PROGRAM P3_03_ProcessData
VAR
	stDBParam 					:ST_ProcessData;	
	fbDBWrite					:FB_PLCDBWriteEvt(sNetId:=CONST.AMS_NETID, tTimeout:=DEFAULT_ADS_TIMEOUT);
	tableColumns				:ARRAY [0..8] OF STRING(50) := ['batch', 'number', 'name', 'value1', 'value2', 'value3', 'value4', 'value5', 'value6'];
	arrParam					:ARRAY [0..8] OF ST_ExpParameter := [(sParaName := 'batch', nParaSize := 101, eParaType := E_EXPPARAMETERTYPE.STRING_),
															 (sParaName := 'number', nParaSize := 101, eParaType := E_EXPPARAMETERTYPE.STRING_),
															 (sParaName := 'name', nParaSize := 101, eParaType := E_EXPPARAMETERTYPE.STRING_),
															 (sParaName := 'value1', nParaSize := 101, eParaType := E_EXPPARAMETERTYPE.Float32), 
															 (sParaName := 'value2', nParaSize := 101, eParaType := E_EXPPARAMETERTYPE.Float32),
															 (sParaName := 'value3', nParaSize := 101, eParaType := E_EXPPARAMETERTYPE.Float32),
															 (sParaName := 'value4', nParaSize := 101, eParaType := E_EXPPARAMETERTYPE.Float32),
															 (sParaName := 'value5', nParaSize := 101, eParaType := E_EXPPARAMETERTYPE.Float32),
															 (sParaName := 'value6', nParaSize := 101, eParaType := E_EXPPARAMETERTYPE.Float32)];
	fbDeleteTable    			:FB_PLCDBCmdEvt(sNetID:=CONST.AMS_NETID, tTimeout:=DEFAULT_ADS_TIMEOUT);	
	sDelete						:STRING;	
	sDeleteAll					:STRING;
	sDeleteBatch				:STRING;
	bDelete						:BOOL;								 
	bWrite						:BOOL;		
	
	rChopper1Speed				:REAL;
	rChopper2Speed				:REAL;
END_VAR
VAR // added by the converter: edge detectors and wires of the graphical bodies
    _rt1, _rt2 : R_TRIG;
END_VAR

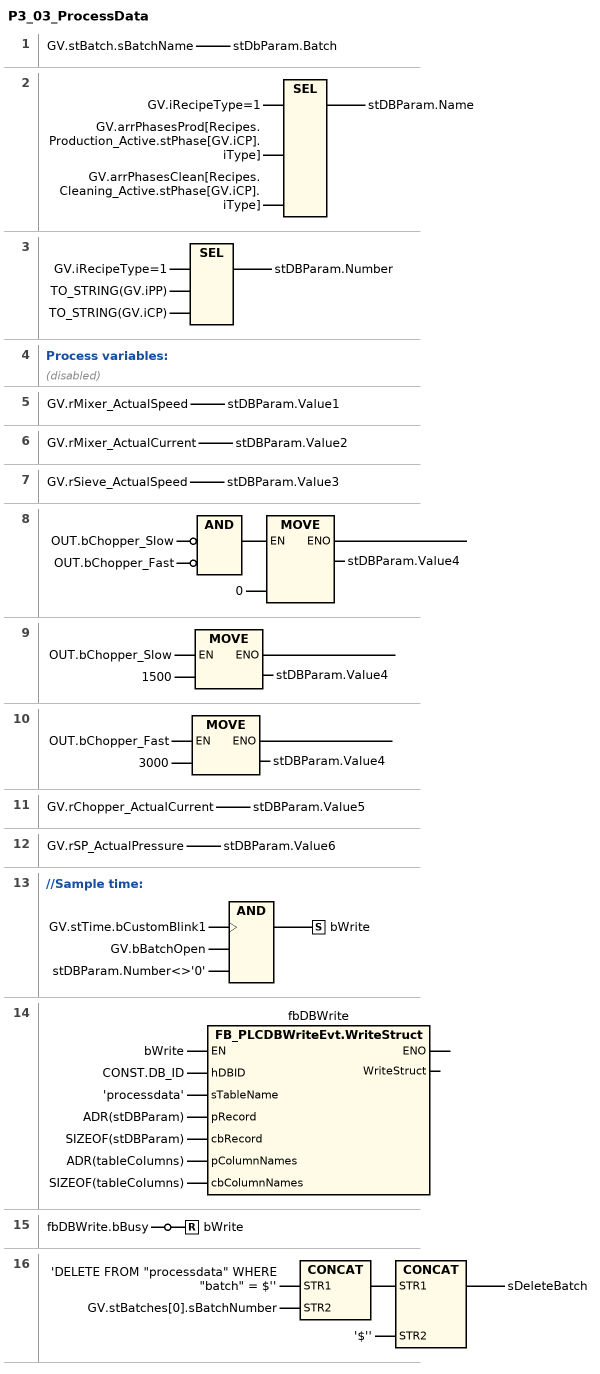
// NETWORK 1
stDbParam.Batch := GV.stBatch.sBatchName;

// NETWORK 2
stDBParam.Name := SEL(GV.iRecipeType=1, GV.arrPhasesProd[Recipes.Production_Active.stPhase[GV.iCP].iType], GV.arrPhasesClean[Recipes.Cleaning_Active.stPhase[GV.iCP].iType]);

// NETWORK 3
stDBParam.Number := SEL(GV.iRecipeType=1, TO_STRING(GV.iPP), TO_STRING(GV.iCP));

// NETWORK 4 (disabled)
// label: Process variables

// NETWORK 5
stDBParam.Value1 := GV.rMixer_ActualSpeed;

// NETWORK 6
stDBParam.Value2 := GV.rMixer_ActualCurrent;

// NETWORK 7
stDBParam.Value3 := GV.rSieve_ActualSpeed;

// NETWORK 8
IF NOT OUT.bChopper_Slow AND NOT OUT.bChopper_Fast THEN stDBParam.Value4 := 0; END_IF

// NETWORK 9
IF OUT.bChopper_Slow THEN stDBParam.Value4 := 1500; END_IF

// NETWORK 10
IF OUT.bChopper_Fast THEN stDBParam.Value4 := 3000; END_IF

// NETWORK 11
stDBParam.Value5 := GV.rChopper_ActualCurrent;

// NETWORK 12
stDBParam.Value6 := GV.rSP_ActualPressure;

// NETWORK 13
// label: //Sample time
_rt1(CLK := GV.stTime.bCustomBlink1);
bWrite S= _rt1.Q AND GV.bBatchOpen AND (stDBParam.Number<>'0');

// NETWORK 14
IF bWrite THEN
    fbDBWrite.WriteStruct(
        hDBID := CONST.DB_ID,
        sTableName := 'processdata',
        pRecord := ADR(stDBParam),
        cbRecord := SIZEOF(stDBParam),
        pColumnNames := ADR(tableColumns),
        cbColumnNames := SIZEOF(tableColumns));
END_IF

// NETWORK 15
bWrite R= NOT fbDBWrite.bBusy;

// NETWORK 16
sDeleteBatch := CONCAT(STR1 := CONCAT(STR1 := 'DELETE FROM "processdata" WHERE "batch" = $'', STR2 := GV.stBatches[0].sBatchNumber), STR2 := '$'');

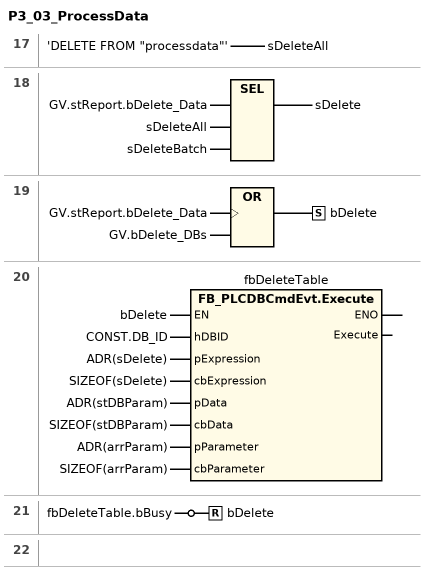
// NETWORK 17
sDeleteAll := 'DELETE FROM "processdata"';

// NETWORK 18
sDelete := SEL(GV.stReport.bDelete_Data, sDeleteAll, sDeleteBatch);

// NETWORK 19
_rt2(CLK := GV.stReport.bDelete_Data);
bDelete S= _rt2.Q OR GV.bDelete_DBs;

// NETWORK 20
IF bDelete THEN
    fbDeleteTable.Execute(
        hDBID := CONST.DB_ID,
        pExpression := ADR(sDelete),
        cbExpression := SIZEOF(sDelete),
        pData := ADR(stDBParam),
        cbData := SIZEOF(stDBParam),
        pParameter := ADR(arrParam),
        cbParameter := SIZEOF(arrParam));
END_IF

// NETWORK 21
bDelete R= NOT fbDeleteTable.bBusy;

// NETWORK 22

END_PROGRAM

(* stored: Version 1.1.0.1, ProductVersion 3.1.4026.13
   POU P3_03_ProcessData: Id {4ea024c6-218b-490f-a3e5-dbb784c2f5cd}, SpecialFunc None *)
